# EPICS substitutions: evrSupport/Db/ioc/IOC-LI25-PM01pattern.substitutions
#
# Pattern records
file evrPatternAll.db {
#	    Device        ,  SLC Pattern Check LNK    , EVR/Trigger
#	                                                  Links
  pattern { DEVICE        ,        LINK4              , LINK5 , LINK6 }
	  { IOC:LI25:PM01 ,         ""                ,  ""   ,  ""   }
}
file evrEventAll.db {
  pattern { DEVICE }
	  { IOC:LI25:PM01}
}
